PROGRAM pouS5Prompts
VAR
	


idbMsgPrompt: FB_CheckMessageBounds;
END_VAR

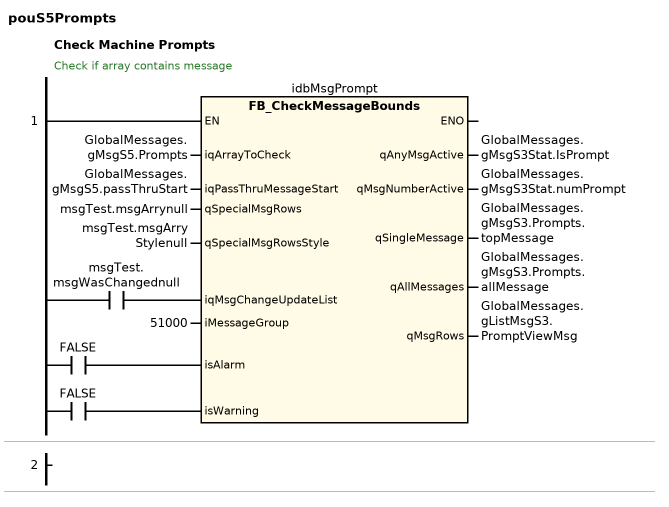
// NETWORK 1: Check Machine Prompts
// Check if array contains message
idbMsgPrompt(
    iqArrayToCheck := GlobalMessages.gMsgS5.Prompts,
    iqPassThruMessageStart := GlobalMessages.gMsgS5.passThruStart,
    qSpecialMsgRows := msgTest.msgArrynull,
    qSpecialMsgRowsStyle := msgTest.msgArryStylenull,
    iqMsgChangeUpdateList := msgTest.msgWasChangednull,
    iMessageGroup := 51000,
    isAlarm := FALSE,
    isWarning := FALSE,
    qAnyMsgActive => GlobalMessages.gMsgS3Stat.IsPrompt,
    qMsgNumberActive => GlobalMessages.gMsgS3Stat.numPrompt,
    qSingleMessage => GlobalMessages.gMsgS3.Prompts.topMessage,
    qAllMessages => GlobalMessages.gMsgS3.Prompts.allMessage,
    qMsgRows => GlobalMessages.gListMsgS3.PromptViewMsg); // FB_CheckMessageBounds

// NETWORK 2

END_PROGRAM

(* stored: Version 1.1.0.1, ProductVersion 3.1.4024.12
   POU pouS5Prompts: Id {bc0bd697-4d36-44ee-a168-cb9bd83cbb84}, SpecialFunc None *)
